FUNCTION_BLOCK PUBLIC Printer
VAR
	 documentType: STRING ;
     sheet: STRING ;
     color : BOOL ;
     text: STRING ;
END_VAR

PROPERTY PUBLIC getDocumentType : STRING
GET
getDocumentType := documentType;
END_GET
END_PROPERTY

PROPERTY PUBLIC getSheet : STRING
GET
getSheet := sheet;
END_GET
END_PROPERTY

PROPERTY PUBLIC getText : STRING
GET
getText := text;
END_GET
END_PROPERTY

PROPERTY PUBLIC isColor : BOOL
GET
isColor := color;
END_GET
END_PROPERTY

METHOD PUBLIC printDocument
VAR
	stext1 : STRING;
	stext2 : STRING;
	stext3 : STRING;
	stext4 : STRING;
	stext : STRING;
	strSFCErrorStep : STRING:='';
END_VAR
//    System.out.println("printing:"+ text+ ",color:"
//        + color+",type:"+DocumentType+",sheet :"+sheet);
		
stext1 := CONCAT(STR1:='printing: ' , STR2:= text);
stext2 := CONCAT(STR1:=', color: ' , STR2:= TO_STRING(color));
stext3 := CONCAT(STR1:=', type: ' , STR2:= DocumentType);
stext4 := CONCAT(STR1:=', sheet: ' , STR2:= sheet);
stext :=  CONCAT(STR1:=stext1 , STR2:=CONCAT(STR1:=stext2 , STR2:=CONCAT(STR1:=stext3 , STR2:=stext4)));
		
 ADSLOGSTR( msgCtrlMask := ADSLOG_MSGTYPE_LOG, msgFmtStr := stext, strArg := strSFCErrorStep);
END_METHOD

METHOD PUBLIC setColor
VAR_INPUT
	color : BOOL;
END_VAR
THIS^.color := color;
END_METHOD

METHOD PUBLIC setDocumentType
VAR_INPUT
	documentType :STRING;
END_VAR
THIS^.documentType := documentType;
END_METHOD

METHOD PUBLIC setSheet
VAR_INPUT
	sheet: STRING ;
END_VAR
THIS^.sheet := sheet;
END_METHOD

METHOD PUBLIC setText
VAR_INPUT
	text :STRING ;
END_VAR
THIS^.text := text;
END_METHOD

END_FUNCTION_BLOCK

(* stored: Version 1.1.0.1, ProductVersion 3.1.4024.12
   POU Printer: Id {387825cd-43cd-4313-84cc-61b0fbf546d4}, SpecialFunc None
   Property getDocumentType: Id {5c1e1859-bb1d-48bb-9345-c0e7db31e48f}
   Get Get: Id {e1cf4236-15da-48ec-a9fb-0b97781c3e0c}
   Property getSheet: Id {0776cd8f-29b0-4d04-8357-e5b6dd51118f}
   Get Get: Id {a0942d40-adde-485e-924f-e0c1c4ef37b5}
   Property getText: Id {d2aa370f-1bf0-4ce7-86c2-5a7f48b420e1}
   Get Get: Id {7f8c68b5-947c-4f93-97ae-4cb59042fa9e}
   Property isColor: Id {260c4854-474f-45d2-87f8-41d36de4859d}
   Get Get: Id {2e2c986a-828a-4dc7-873c-8c42e5247795}
   Method printDocument: Id {bc84cfcc-1995-4d28-8554-ab0463361273}
   Method setColor: Id {0826e445-6054-430b-9928-a71926c5d035}
   Method setDocumentType: Id {18dc93e2-08bc-4aa0-81b5-d04ff55f4bba}
   Method setSheet: Id {392a0520-49f7-4240-bf11-3d53aebe630c}
   Method setText: Id {d2e32e99-6553-46e7-b954-e306a5ee30f5} *)
